// TIA Portal V18 export
TYPE "IAI Output Struct"
   STRUCT
      "Output 4 word_Man1" : Struct
         "Reserve_0.0" : Bool;
         "Reserve_0.1" : Bool;
         "Reserve_0.2" : Bool;
         "Reserve_0.3" : Bool;
         "Reserve_0.4" : Bool;
         "Reserve_0.5" : Bool;
         "Reserve_0.6" : Bool;
         Mon : Bool;   // PLC控制输出有效
         Reserve_1 : Byte;
         Reserve_2 : Int;
         Reserve_4 : Int;
         Reserve_6 : Int;
      END_STRUCT;
      "Output 4 word_Man2" : Struct
         Reserve_8 : Int;
         Reserve_10 : Int;
         Reserve_12 : Int;
         Reserve_14 : Int;
      END_STRUCT;
      "Output 4 word_1" : Struct
         "Target position" : DInt;
         "Location Width" : DInt;
      END_STRUCT;
      "Output 4 word_2" : Struct
         Speed : Int;
         "Accelerated Speed" : Int;   // 加速度
         "Push Current" : Int;   // 推压时电流限制值
         "JOG+" : Bool;   // ＋JOG
         Spare_1 : Bool;   // 不能使用
         Spare_2 : Bool;   // 不能使用
         Spare_3 : Bool;   // 不能使用
         Push : Bool;   // 推压指定
         DIR : Bool;   // 推压方向指定
         INC : Bool;   // 增量型
         BKRL : Bool;   // 刹车强制解除
         CSTR : Bool;   // 定位开始
         Home : Bool;   // 原点复位
         STP : Bool;   // 暂停
         RES : Bool;   // 复位
         SON : Bool;   // 伺服ON指令
         JISL : Bool;   // JOG/微调切换
         JVEL : Bool;   // JOG速度/微调距离切换
         "JOG-" : Bool;   // －JOG
      END_STRUCT;
   END_STRUCT;
END_TYPE
